PROGRAM LM_State_MC_TCP
VAR
END_VAR

// NETWORK 1

END_PROGRAM

(* stored: Version 1.1.0.1, ProductVersion 3.1.4024.0
   POU LM_State_MC_TCP: Id {a40c49c4-0a92-49ee-86d6-e0e524236872}, SpecialFunc None *)
